TYPE ST_KPI_OutersProcessing :
STRUCT
	AtPackAggregCameras	: UDINT;
	AtConfimrationCamera 	: UDINT;
	AtValidationCamera		: UDINT;
END_STRUCT
END_TYPE

(* stored: Version 1.1.0.1, ProductVersion 3.1.4024.15
   DUT ST_KPI_OutersProcessing: Id {b6f4bdf8-86fd-453f-b94e-55f64bf4cdd3} *)
